Omron CX-Programmer project NouvProjet (CX-Programmer 9.61)

# PLC NouvAPI1: CP1L M

## Global symbols (name address type ; comment)
0.00 BOOL  ; Reset
0.01 BOOL  ; m1
0.02 BOOL  ; m2
0.03 BOOL  ; a1
0.04 BOOL  ; a2
0.05 BOOL  ; AU
0.06 BOOL  ; SPDATK
0.07 BOOL  ; SPGATK
0.08 BOOL  ; CVATK
0.09 BOOL  ; SPDFBK
0.10 BOOL  ; SPGFBK
0.11 BOOL  ; Q1+F7
100.00 BOOL  ; KM1
100.01 BOOL  ; KM4
100.02 BOOL  ; KM5.1M9
100.03 BOOL  ; KM9
100.04 BOOL  ; KM8
100.05 BOOL  ; FBK
100.06 BOOL  ; Y5
100.07 BOOL  ; V1
101.00 BOOL  ; V2
101.01 BOOL  ; V3
101.02 BOOL  ; V4
101.03 BOOL  ; Lampe de Signalisation
10.00 BOOL  ; X0
10.01 BOOL  ; X1
10.02 BOOL  ; X2
10.03 BOOL  ; X3
10.04 BOOL  ; X4
10.05 BOOL  ; X5
10.06 BOOL  ; X6
10.07 BOOL  ; X7
10.08 BOOL  ; X8
10.09 BOOL  ; X9
10.10 BOOL  ; X10
10.11 BOOL  ; X11
10.12 BOOL  ; X12
10.13 BOOL  ; X13
1.00 BOOL  ; F1+F2+Q4+Q5+Q20
1.01 BOOL  ; Q10+Q11+F3
1.02 BOOL  ; B7+B8
1.03 BOOL  ; Bouton
1.04 BOOL  ; Commutateur
200.00 BOOL  ; Init
20.00 BOOL  ; X20
20.01 BOOL  ; X21
20.02 BOOL  ; X22
20.03 BOOL  ; X23
20.04 BOOL  ; X24
20.05 BOOL  ; X25
30.00 BOOL  ; X30
30.01 BOOL  ; X31
40.00 BOOL  ; X40
40.01 BOOL  ; X41
80.00 BOOL  ; Chaine de securité ATK
80.01 BOOL  ; Chaine de securité FBK
80.02 BOOL  ; Chaine  des défauts

## Program NouvProgramme1 (cyclic task 0)

### Section Programmation_d_une_Machine_de_cardage

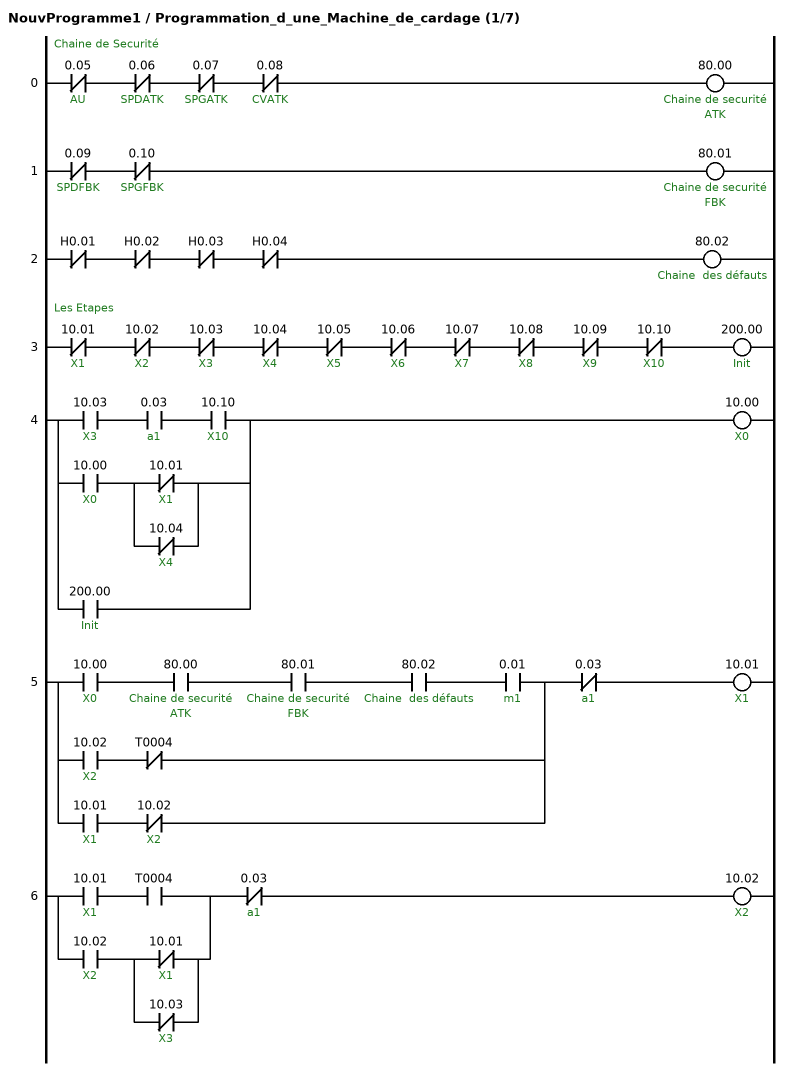
; rung 0: Chaine de Securité
LDNOT 0.05  ; AU
ANDNOT 0.06  ; SPDATK
ANDNOT 0.07  ; SPGATK
ANDNOT 0.08  ; CVATK
OUT 80.00  ; Chaine de securité ATK
; rung 1
LDNOT 0.09  ; SPDFBK
ANDNOT 0.10  ; SPGFBK
OUT 80.01  ; Chaine de securité FBK
; rung 2
LDNOT H0.01
ANDNOT H0.02
ANDNOT H0.03
ANDNOT H0.04
OUT 80.02  ; Chaine  des défauts
; rung 3: Les Etapes
LDNOT 10.01  ; X1
ANDNOT 10.02  ; X2
ANDNOT 10.03  ; X3
ANDNOT 10.04  ; X4
ANDNOT 10.05  ; X5
ANDNOT 10.06  ; X6
ANDNOT 10.07  ; X7
ANDNOT 10.08  ; X8
ANDNOT 10.09  ; X9
ANDNOT 10.10  ; X10
OUT 200.00  ; Init
; rung 4
LD 10.03  ; X3
AND 0.03  ; a1
AND 10.10  ; X10
LD 10.00  ; X0
LDNOT 10.01  ; X1
ORNOT 10.04  ; X4
ANDLD
ORLD
OR 200.00  ; Init
OUT 10.00  ; X0
; rung 5
LD 10.00  ; X0
AND 80.00  ; Chaine de securité ATK
AND 80.01  ; Chaine de securité FBK
AND 80.02  ; Chaine  des défauts
AND 0.01  ; m1
LD 10.02  ; X2
ANDNOT T0004
ORLD
LD 10.01  ; X1
ANDNOT 10.02  ; X2
ORLD
ANDNOT 0.03  ; a1
OUT 10.01  ; X1
; rung 6
LD 10.01  ; X1
AND T0004
LD 10.02  ; X2
LDNOT 10.01  ; X1
ORNOT 10.03  ; X3
ANDLD
ORLD
ANDNOT 0.03  ; a1
OUT 10.02  ; X2

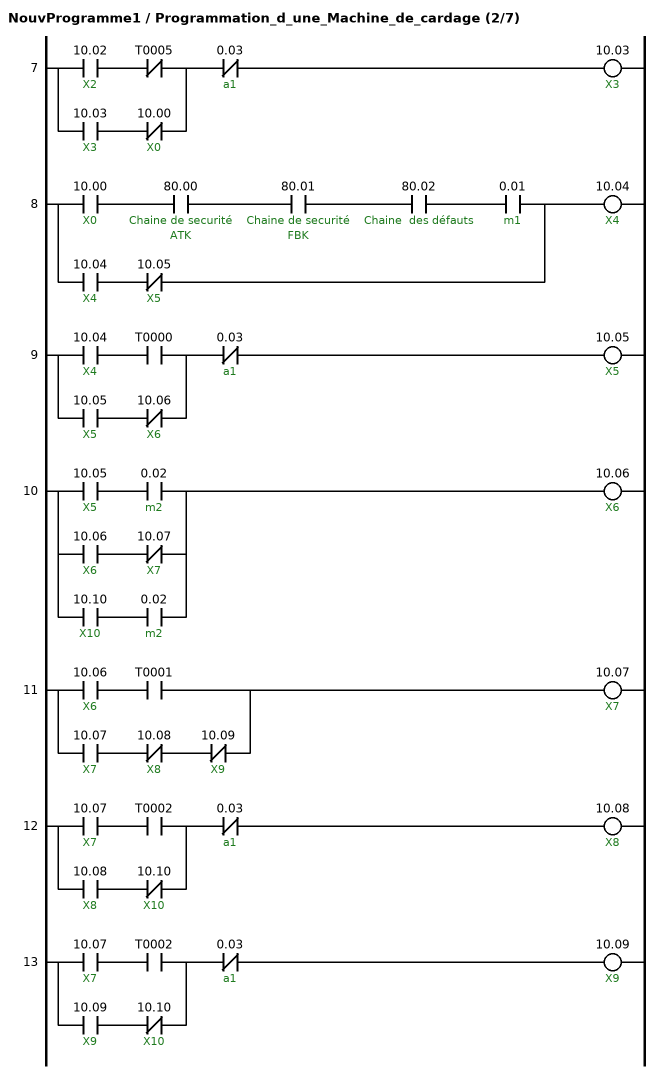
; rung 7
LD 10.02  ; X2
ANDNOT T0005
LD 10.03  ; X3
ANDNOT 10.00  ; X0
ORLD
ANDNOT 0.03  ; a1
OUT 10.03  ; X3
; rung 8
LD 10.00  ; X0
AND 80.00  ; Chaine de securité ATK
AND 80.01  ; Chaine de securité FBK
AND 80.02  ; Chaine  des défauts
AND 0.01  ; m1
LD 10.04  ; X4
ANDNOT 10.05  ; X5
ORLD
OUT 10.04  ; X4
; rung 9
LD 10.04  ; X4
AND T0000
LD 10.05  ; X5
ANDNOT 10.06  ; X6
ORLD
ANDNOT 0.03  ; a1
OUT 10.05  ; X5
; rung 10
LD 10.05  ; X5
AND 0.02  ; m2
LD 10.06  ; X6
ANDNOT 10.07  ; X7
ORLD
LD 10.10  ; X10
AND 0.02  ; m2
ORLD
OUT 10.06  ; X6
; rung 11
LD 10.06  ; X6
AND T0001
LD 10.07  ; X7
ANDNOT 10.08  ; X8
ANDNOT 10.09  ; X9
ORLD
OUT 10.07  ; X7
; rung 12
LD 10.07  ; X7
AND T0002
LD 10.08  ; X8
ANDNOT 10.10  ; X10
ORLD
ANDNOT 0.03  ; a1
OUT 10.08  ; X8
; rung 13
LD 10.07  ; X7
AND T0002
LD 10.09  ; X9
ANDNOT 10.10  ; X10
ORLD
ANDNOT 0.03  ; a1
OUT 10.09  ; X9

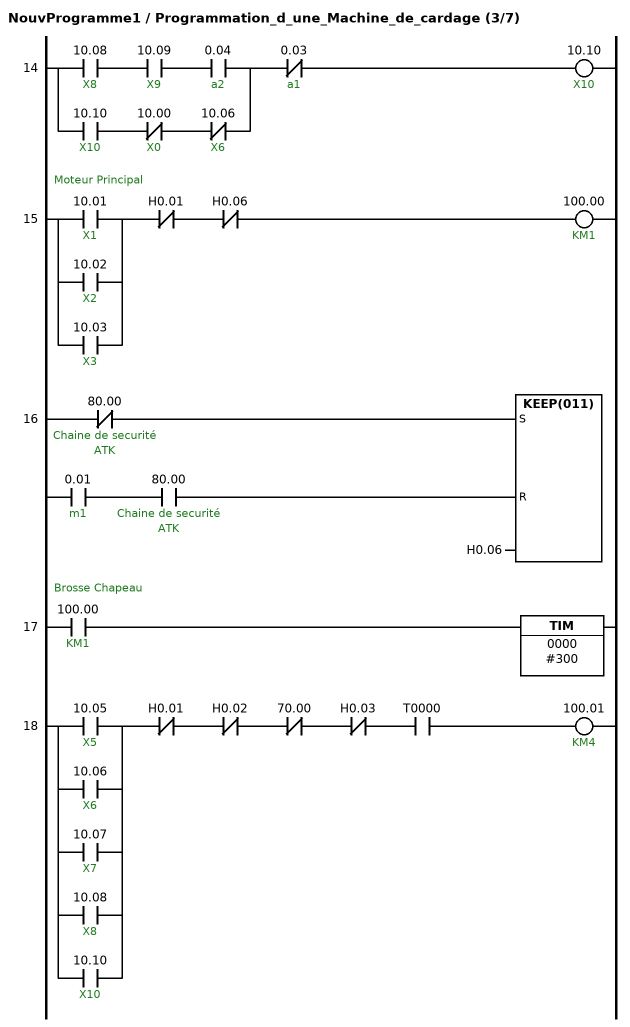
; rung 14
LD 10.08  ; X8
AND 10.09  ; X9
AND 0.04  ; a2
LD 10.10  ; X10
ANDNOT 10.00  ; X0
ANDNOT 10.06  ; X6
ORLD
ANDNOT 0.03  ; a1
OUT 10.10  ; X10
; rung 15: Moteur Principal
LD 10.01  ; X1
OR 10.02  ; X2
OR 10.03  ; X3
ANDNOT H0.01
ANDNOT H0.06
OUT 100.00  ; KM1
; rung 16
LDNOT 80.00  ; Chaine de securité ATK
LD 0.01  ; m1
AND 80.00  ; Chaine de securité ATK
KEEP(011) H0.06
; rung 17: Brosse Chapeau
LD 100.00  ; KM1
TIM 0000 #300
; rung 18
LD 10.05  ; X5
OR 10.06  ; X6
OR 10.07  ; X7
OR 10.08  ; X8
OR 10.10  ; X10
ANDNOT H0.01
ANDNOT H0.02
ANDNOT 70.00
ANDNOT H0.03
AND T0000
OUT 100.01  ; KM4

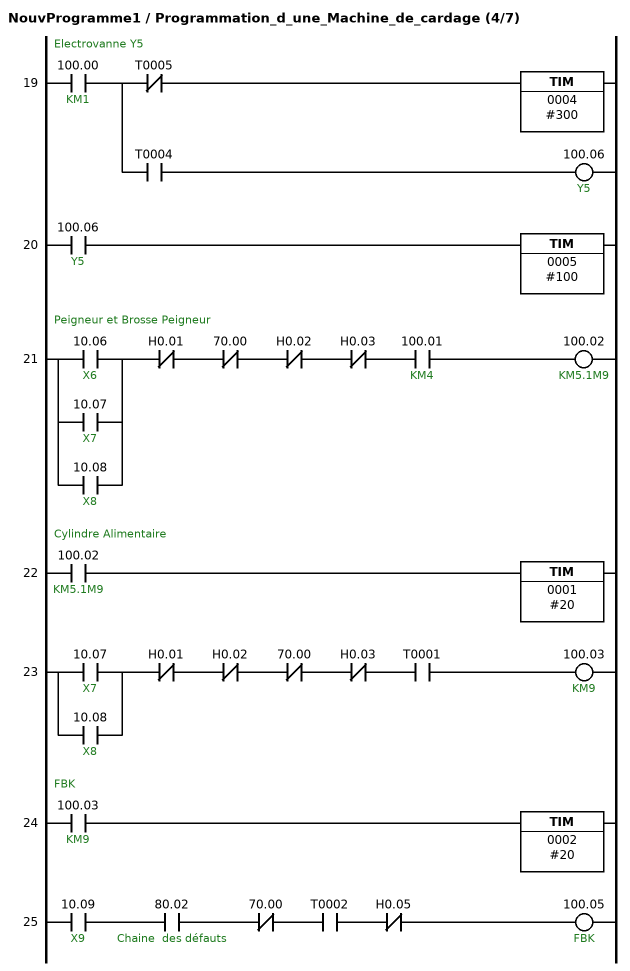
; rung 19: Electrovanne Y5
LD 100.00  ; KM1
OUT TR0
ANDNOT T0005
TIM 0004 #300
LD TR0
AND T0004
OUT 100.06  ; Y5
; rung 20
LD 100.06  ; Y5
TIM 0005 #100
; rung 21: Peigneur et Brosse Peigneur
LD 10.06  ; X6
OR 10.07  ; X7
OR 10.08  ; X8
ANDNOT H0.01
ANDNOT 70.00
ANDNOT H0.02
ANDNOT H0.03
AND 100.01  ; KM4
OUT 100.02  ; KM5.1M9
; rung 22: Cylindre Alimentaire
LD 100.02  ; KM5.1M9
TIM 0001 #20
; rung 23
LD 10.07  ; X7
OR 10.08  ; X8
ANDNOT H0.01
ANDNOT H0.02
ANDNOT 70.00
ANDNOT H0.03
AND T0001
OUT 100.03  ; KM9
; rung 24: FBK
LD 100.03  ; KM9
TIM 0002 #20
; rung 25
LD 10.09  ; X9
AND 80.02  ; Chaine  des défauts
ANDNOT 70.00
AND T0002
ANDNOT H0.05
OUT 100.05  ; FBK

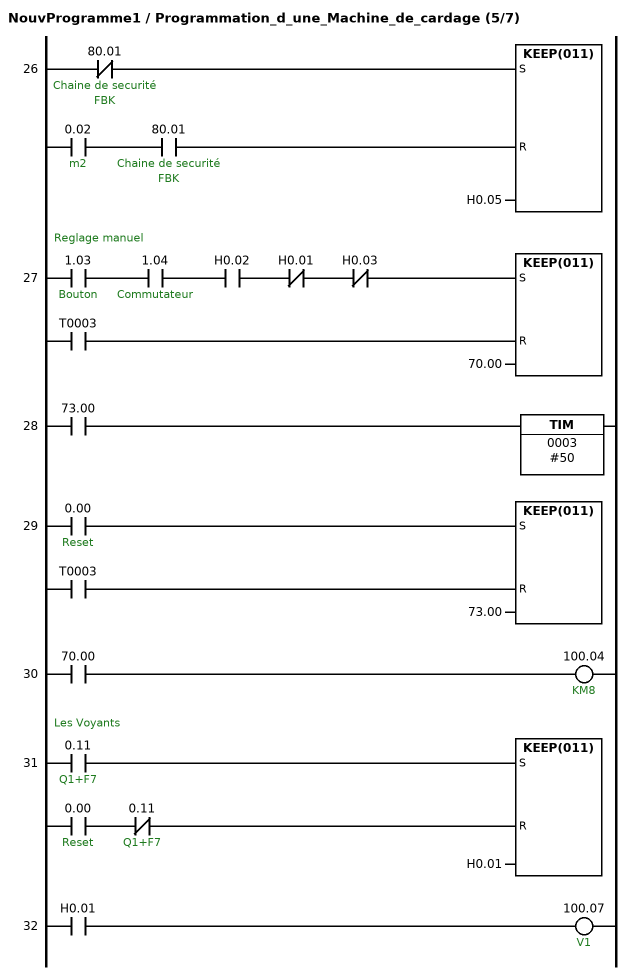
; rung 26
LDNOT 80.01  ; Chaine de securité FBK
LD 0.02  ; m2
AND 80.01  ; Chaine de securité FBK
KEEP(011) H0.05
; rung 27: Reglage manuel
LD 1.03  ; Bouton
AND 1.04  ; Commutateur
AND H0.02
ANDNOT H0.01
ANDNOT H0.03
LD T0003
KEEP(011) 70.00
; rung 28
LD 73.00
TIM 0003 #50
; rung 29
LD 0.00  ; Reset
LD T0003
KEEP(011) 73.00
; rung 30
LD 70.00
OUT 100.04  ; KM8
; rung 31: Les Voyants
LD 0.11  ; Q1+F7
LD 0.00  ; Reset
ANDNOT 0.11  ; Q1+F7
KEEP(011) H0.01
; rung 32
LD H0.01
OUT 100.07  ; V1

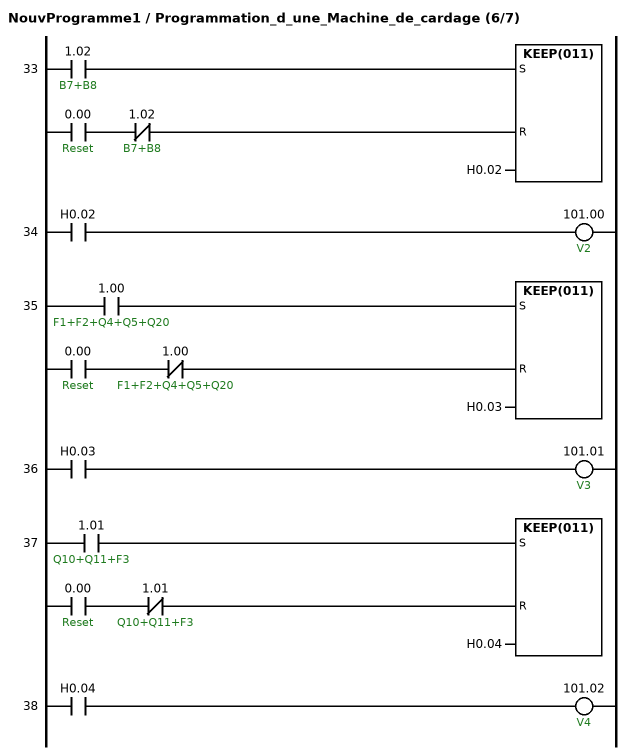
; rung 33
LD 1.02  ; B7+B8
LD 0.00  ; Reset
ANDNOT 1.02  ; B7+B8
KEEP(011) H0.02
; rung 34
LD H0.02
OUT 101.00  ; V2
; rung 35
LD 1.00  ; F1+F2+Q4+Q5+Q20
LD 0.00  ; Reset
ANDNOT 1.00  ; F1+F2+Q4+Q5+Q20
KEEP(011) H0.03
; rung 36
LD H0.03
OUT 101.01  ; V3
; rung 37
LD 1.01  ; Q10+Q11+F3
LD 0.00  ; Reset
ANDNOT 1.01  ; Q10+Q11+F3
KEEP(011) H0.04
; rung 38
LD H0.04
OUT 101.02  ; V4

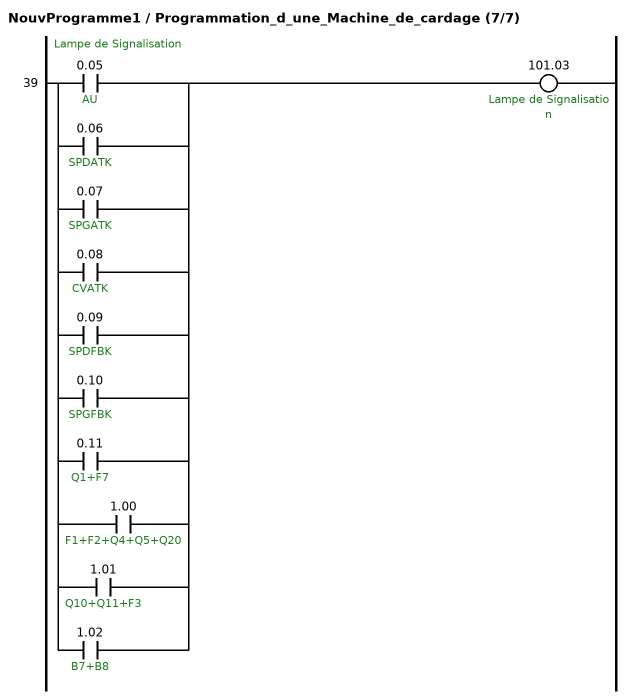
; rung 39: Lampe de Signalisation
LD 0.05  ; AU
OR 0.06  ; SPDATK
OR 0.07  ; SPGATK
OR 0.08  ; CVATK
OR 0.09  ; SPDFBK
OR 0.10  ; SPGFBK
OR 0.11  ; Q1+F7
OR 1.00  ; F1+F2+Q4+Q5+Q20
OR 1.01  ; Q10+Q11+F3
OR 1.02  ; B7+B8
OUT 101.03  ; Lampe de Signalisation

### Section END
; rung 0
END(001)